// TIA Portal V19 export
VAR_GLOBAL   // PLC tag table "Default tag table"
   memstart1 AT %M2.2 : Bool;
END_VAR
